// TIA Portal V17 export
// export: Created 2023-02-26T22:59:49.8656164Z, ExportSetting WithDefaults, DisplayName Totally Integrated Automation Portal, DisplayVersion V17, DisplayName TIA Portal Openness, DisplayVersion V17, DisplayName TIA Portal Version Control Interface, DisplayVersion V17, DisplayName TIA Portal Test Suite Advanced, DisplayVersion V17, DisplayName STEP 7 Professional, DisplayVersion V17, DisplayName SIMATIC Energy Suite, DisplayVersion V17, DisplayName STEP 7 Safety, DisplayVersion V17, DisplayName WinCC Professional, DisplayVersion V17
FUNCTION "LOG_CalculateWorkTime" : Void   // FC1300, LAD
{ S7_Optimized_Access := 'TRUE' }
VERSION : 0.1
// stored: AutoNumber false, IsIECCheckEnabled false, SetENOAutomatically false, UDAEnableTagReadback false
   VAR_INPUT
      Trigger : Bool;
   END_VAR
   VAR_IN_OUT
      LineTime : "stt_TimeWork";
   END_VAR
   VAR_TEMP   // added for the SCL form of the ladder/FBD networks
      _w1 : Bool;
   END_VAR
BEGIN

REGION Network 1: Seconds
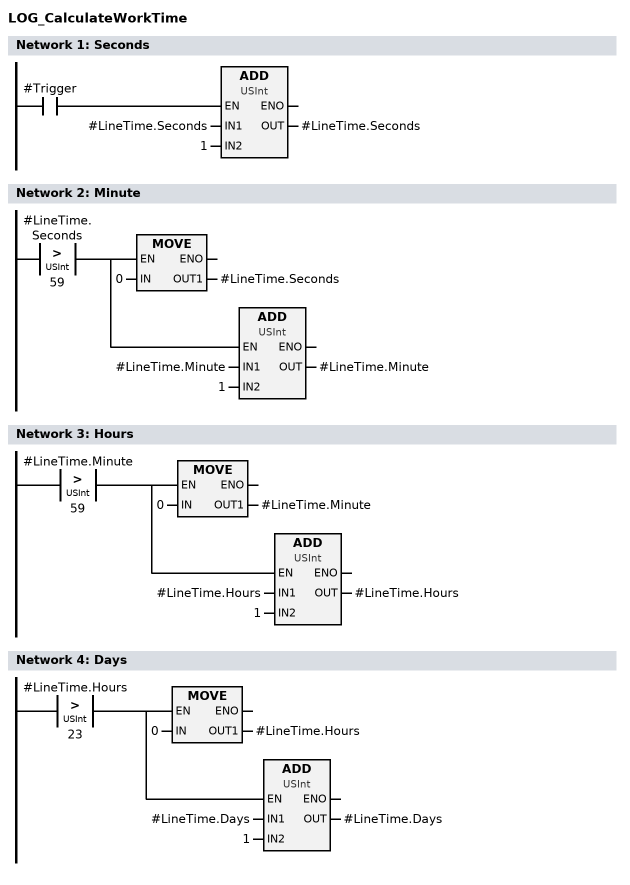
   RUNG wire#powerrail
      Contact( #Trigger )
      { S7_Templates := "SrcType := USInt"; S7_GenerateENO := "TRUE" } Add(in1 := #LineTime.Seconds, in2 := 1, out => #LineTime.Seconds)
   END_RUNG
   // the same network as SCL:
   IF #Trigger THEN #LineTime.Seconds := #LineTime.Seconds + 1; END_IF;
END_REGION

REGION Network 2: Minute
   RUNG wire#powerrail
      { S7_Templates := "SrcType := USInt" } GT_Contact(in1 := #LineTime.Seconds, in2 := 59)
      wire#w1
      { S7_GenerateENO := "TRUE" } Move(in := 0, out1 => #LineTime.Seconds)
   END_RUNG
   RUNG wire#w1
      { S7_Templates := "SrcType := USInt"; S7_GenerateENO := "TRUE" } Add(in1 := #LineTime.Minute, in2 := 1, out => #LineTime.Minute)
   END_RUNG
   // the same network as SCL:
   #_w1 := #LineTime.Seconds > 59;
   IF #_w1 THEN
       #LineTime.Seconds := 0;
       #LineTime.Minute := #LineTime.Minute + 1;
   END_IF;
END_REGION

REGION Network 3: Hours
   RUNG wire#powerrail
      { S7_Templates := "SrcType := USInt" } GT_Contact(in1 := #LineTime.Minute, in2 := 59)
      wire#w1
      { S7_GenerateENO := "TRUE" } Move(in := 0, out1 => #LineTime.Minute)
   END_RUNG
   RUNG wire#w1
      { S7_Templates := "SrcType := USInt"; S7_GenerateENO := "TRUE" } Add(in1 := #LineTime.Hours, in2 := 1, out => #LineTime.Hours)
   END_RUNG
   // the same network as SCL:
   #_w1 := #LineTime.Minute > 59;
   IF #_w1 THEN
       #LineTime.Minute := 0;
       #LineTime.Hours := #LineTime.Hours + 1;
   END_IF;
END_REGION

REGION Network 4: Days
   RUNG wire#powerrail
      { S7_Templates := "SrcType := USInt" } GT_Contact(in1 := #LineTime.Hours, in2 := 23)
      wire#w1
      { S7_GenerateENO := "TRUE" } Move(in := 0, out1 => #LineTime.Hours)
   END_RUNG
   RUNG wire#w1
      { S7_Templates := "SrcType := USInt"; S7_GenerateENO := "TRUE" } Add(in1 := #LineTime.Days, in2 := 1, out => #LineTime.Days)
   END_RUNG
   // the same network as SCL:
   #_w1 := #LineTime.Hours > 23;
   IF #_w1 THEN
       #LineTime.Hours := 0;
       #LineTime.Days := #LineTime.Days + 1;
   END_IF;
END_REGION
END_FUNCTION
